Fanuc KAREL source: VT_GET_TRYID.kl

PROGRAM T
%NOLOCKGROUP
VAR
 v0 : STRING[40]
 res : INTEGER
BEGIN
 res = VT_GET_TRYID(v0)
END T
